(* PLC project Unbenannt1, Beckhoff Automation GmbH TwinCAT PLC Control 3.5.6.1 *)
(* stored: creationDateTime 2016-01-19T13:20:20.3046228, modificationDateTime 2016-01-19T13:20:20.3046228 *)

(* global variable list GVL_Checks *)
VAR_GLOBAL
	CheckBounds_ErrCnt				:DINT;
	CheckDivDInt_ErrCnt				:DINT;
	CheckDivLInt_ErrCnt				:DINT;
	CheckDivLReal_ErrCnt			:DINT;
	CheckDivReal_ErrCnt				:DINT;
	CheckRangeSigned_ErrCnt			:DINT;
	CheckRangeUnsigned_ErrCnt		:DINT;
	
END_VAR

// Implicitly generated code : DO NOT EDIT
FUNCTION CheckBounds : DINT
VAR_INPUT
	index, lower, upper: DINT;
END_VAR

            // Implicitly generated code : Only an Implementation suggestion
IF  index < lower THEN
	CheckBounds := lower;
	CheckBounds_ErrCnt:=CheckBounds_ErrCnt+1;
ELSIF  index > upper THEN
	CheckBounds := upper;
	CheckBounds_ErrCnt:=CheckBounds_ErrCnt+1;
ELSE  
	CheckBounds := index;
END_IF

          
END_FUNCTION

// Implicitly generated code : DO NOT EDIT
FUNCTION CheckDivDInt : DINT
VAR_INPUT
	divisor:DINT;
END_VAR

            // Implicitly generated code : Only an Implementation suggestion
IF divisor = 0 THEN
	CheckDivDInt:=1;
	CheckDivDInt_ErrCnt:=CheckDivDInt_ErrCnt+1;
ELSE
	CheckDivDInt:=divisor;
END_IF;
          
END_FUNCTION

// Implicitly generated code : DO NOT EDIT
FUNCTION CheckDivLInt : LINT
VAR_INPUT
	divisor:LINT;
END_VAR

            // Implicitly generated code : Only an Implementation suggestion
IF divisor = 0 THEN
	CheckDivLInt:=1;
	CheckDivLInt_ErrCnt:=CheckDivLInt_ErrCnt+1;
ELSE
	CheckDivLInt:=divisor;
END_IF;
          
END_FUNCTION

// Implicitly generated code : DO NOT EDIT
FUNCTION CheckDivLReal : LREAL
VAR_INPUT
	divisor:LREAL;
END_VAR

            // Implicitly generated code : Only an Implementation suggestion
IF divisor = 0 THEN
	CheckDivLReal:=1;
	CheckDivLReal_ErrCnt:=CheckDivLReal_ErrCnt+1;
ELSE
	CheckDivLReal:=divisor;
END_IF;
          
END_FUNCTION

// Implicitly generated code : DO NOT EDIT
FUNCTION CheckDivReal : REAL
VAR_INPUT
	divisor:REAL;
END_VAR

            // Implicitly generated code : Only an Implementation suggestion
IF divisor = 0 THEN
	CheckDivReal:=1;
	CheckDivReal_ErrCnt:=CheckDivReal_ErrCnt+1;
ELSE
	CheckDivReal:=divisor;
END_IF;
          
END_FUNCTION

// Implicitly generated code : DO NOT EDIT
FUNCTION CheckPointer : POINTER TO BYTE
VAR_INPUT 
	ptToTest : POINTER TO BYTE; // Destination address of the pointer
	iSize : DINT;		        // Size of the type the pointer points to. (e.g: 20 for POINTER TO ARRAY [0..9] OF INT) 
	iGran : DINT;		        // Granularity of the pointer access. This is the size of the biggest non-structured data type in the type the pointer points to. (e.g: 2 for POINTER TO ARRAY [0..9] OF INT)
	bWrite: BOOL;		        // Indicates read or write Access. TRUE = write access.
END_VAR

            // No standard way of implementation. Fill your own code here
CheckPointer := ptToTest;
          
END_FUNCTION

// Implicitly generated code : DO NOT EDIT
FUNCTION CheckRangeSigned : DINT
VAR_INPUT
	value, lower, upper: DINT;
END_VAR

            // Implicitly generated code : Only an Implementation suggestion
IF (value < lower) THEN
	CheckRangeSigned := lower;
	CheckRangeSigned_ErrCnt:=CheckRangeSigned_ErrCnt+1;
ELSIF(value > upper) THEN
	CheckRangeSigned := upper;
	CheckRangeSigned_ErrCnt:=CheckRangeSigned_ErrCnt+1;
ELSE
	CheckRangeSigned := value;
END_IF
          
END_FUNCTION

// Implicitly generated code : DO NOT EDIT
FUNCTION CheckRangeUnsigned : UDINT
VAR_INPUT
	value, lower, upper: UDINT;
END_VAR

            // Implicitly generated code : Only an Implementation suggestion
IF (value < lower) THEN
	CheckRangeUnsigned := lower;
	CheckRangeUnsigned_ErrCnt:=CheckRangeUnsigned_ErrCnt+1;
ELSIF(value > upper) THEN
	CheckRangeUnsigned := upper;
	CheckRangeUnsigned_ErrCnt:=CheckRangeUnsigned_ErrCnt+1;
ELSE
	CheckRangeUnsigned := value;
END_IF
          
END_FUNCTION
